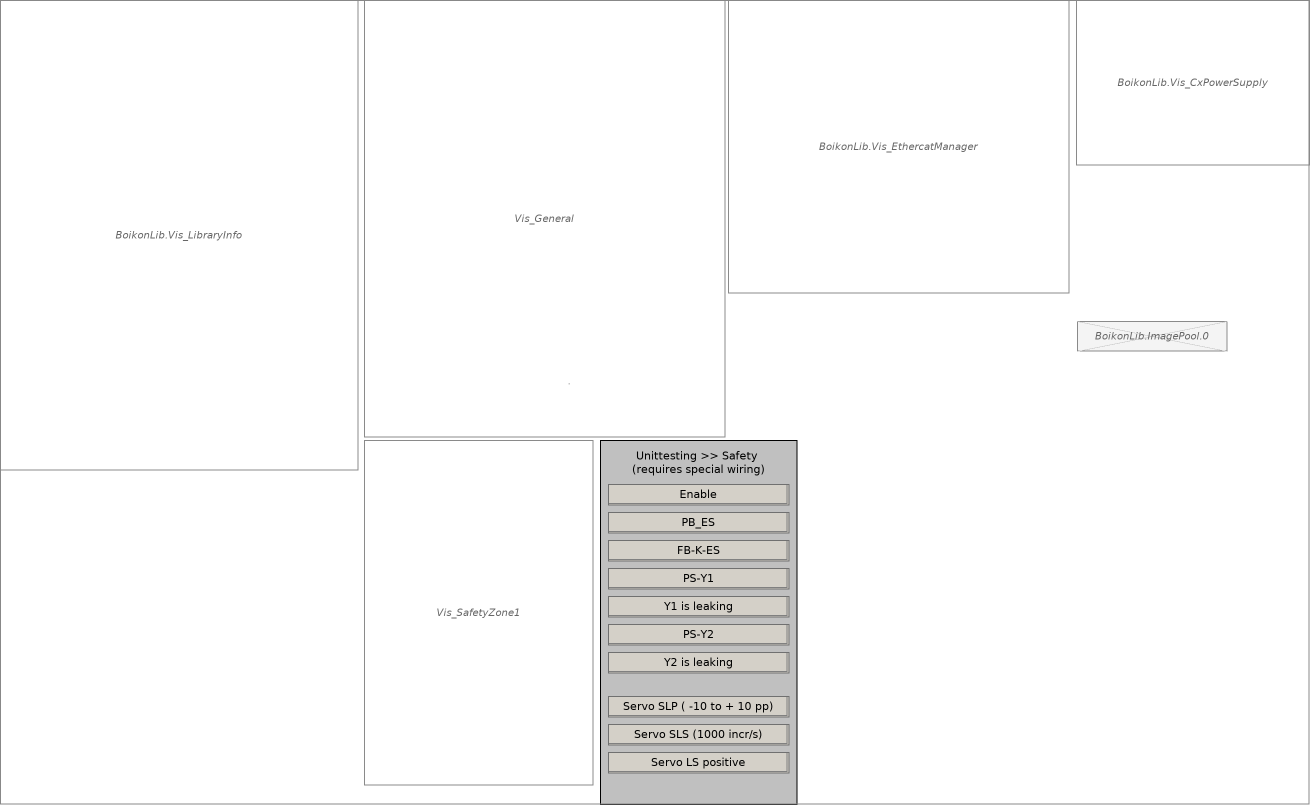
VISUALIZATION VisGeneral  // 1310x805, background image BoikonLib.Images.0
    Rectangle (600,440 197x365)
    Frame (364,0 361x437)
        shows Vis_General(IO_General := MAIN.General)
    Frame (728,0 341x293)
        shows BoikonLib.Vis_EthercatManager(IO_EM := MAIN.General.EthercatManager)
    Frame (364,440 229x345)
        shows Vis_SafetyZone1(I_Title := 'SafetyZone 1', IO_SafetyLogic := MAIN.General.SafetyZone1)
    Frame (1076,0 234x165)
        shows BoikonLib.Vis_CxPowerSupply(I_Title := 'cx power supply', IO := MAIN.General.CxPowerSupply)
    Frame (0,0 358x470)
        shows BoikonLib.Vis_LibraryInfo(IO_Cntrl := MAIN.General.BknLibrary)
    Button (608,540 181x21), "FB-K-ES", pressed state: UnitTesting.Sft_FB_K_ES_OK
        toggle UnitTesting.Sft_FB_K_ES_OK
    Button (608,568 181x21), "PS-Y1", pressed state: UnitTesting.Sft_Y_FB1
        toggle UnitTesting.Sft_Y_FB1
    Button (608,624 181x21), "PS-Y2", pressed state: UnitTesting.Sft_Y_FB2
        toggle UnitTesting.Sft_Y_FB2
    Button (608,512 181x21), "PB_ES", pressed state: UnitTesting.Sft_PB_ES
        toggle UnitTesting.Sft_PB_ES
    Button (608,484 181x21), "Enable", pressed state: UnitTesting.EnableSafetyTest
        toggle UnitTesting.EnableSafetyTest
    Button (608,596 181x21), "Y1 is leaking", pressed state: UnitTesting.Sft_Y1_Leaking
        toggle UnitTesting.Sft_Y1_Leaking
    Button (608,652 181x21), "Y2 is leaking", pressed state: UnitTesting.Sft_Y2_Leaking
        toggle UnitTesting.Sft_Y2_Leaking
    Rectangle (600,440 197x45), "Unittesting >> Safety (requires special wiring)"
    Button (608,696 181x21), "Servo SLP ( -10 to + 10 pp)", pressed state: UnitTesting.Qsf_K_EnableSafePosition
        toggle UnitTesting.Qsf_K_EnableSafePosition
    Button (608,724 181x21), "Servo SLS (1000 incr/s)", pressed state: UnitTesting.Qsf_K_EnableSafeSpeed
        toggle UnitTesting.Qsf_K_EnableSafeSpeed
    Image (569,383 0x1), image: BoikonLib.ImagePool.0
    Button (608,752 181x21), "Servo LS positive", pressed state: UnitTesting.LS_Positive.I_K_State
        toggle UnitTesting.LS_Positive.I_K_State
    Image (1077,321 150x30), image: BoikonLib.ImagePool.0
END_VISUALIZATION

(* stored: Version 1.1.0.1
   Visu VisGeneral: Id {dc8989f6-7b30-4270-87f9-adb84d276bde} *)
